FUNCTION_BLOCK AB_TO_AUDI (* Composite FB for converting AB (BYTE) adapter to AUDI (UDINT) adapter — bit-reinterpretation, value-preserving (destination is same width or wider than the source bit-string). *)
  (* Standard: 61499-2; Description: Copyright (c) 2026 HR Agrartechnik GmbH This program and the accompanying materials are made available under the terms of the Eclipse Public License 2.0 which is available at https://www.eclipse.org/legal/epl-2.0/ SPDX-License-Identifier: EPL-2.0 *)
  (* Version 1.0, 2026-02-17, Franz Höpfinger, HR Agrartechnik GmbH *)
  PACKAGE adapter::conversion::unidirectional;
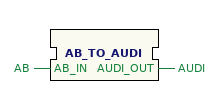
  SOCKETS
    AB_IN : adapter::types::unidirectional::AB; (* BYTE Adapter Input *)
  END_SOCKETS
  PLUGS
    AUDI_OUT : adapter::types::unidirectional::AUDI; (* UDINT Adapter Output *)
  END_PLUGS
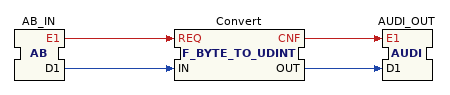
  FBS
    Convert : iec61131::conversion::F_BYTE_TO_UDINT;
  END_FBS
  EVENT_CONNECTIONS
    AB_IN.E1 TO Convert.REQ;
    Convert.CNF TO AUDI_OUT.E1;
  END_CONNECTIONS
  DATA_CONNECTIONS
    AB_IN.D1 TO Convert.IN;
    Convert.OUT TO AUDI_OUT.D1;
  END_CONNECTIONS
END_FUNCTION_BLOCK
